FUNCTION F_ITC_SendFCR : BOOL
(**************************************************************************************
 * 	Application		:	BoxControl Framework
 *	Revision		:	$Revision: 404529 $
 *	Revision date	:	$Date: 2018-04-23 08:21:38 +0200 (Mo., 23 Apr 2018) $
 *	Last changed by	:	$Author: b7bolm $
 *	URL				:	$URL: http://almscdc.swisslog.com/repo/SWPD/Development/BoxControlFramework/20_Release/trunk/01_Software/BCF/BCF/JumpStart/20_Product/10_App/11_Com/10_Lib/10_Conv/11_ITC/F_ITC_SendFCR.TcPOU $
 *
 *	Purpose			:	Wrap message - FCR
 *
 * ------------------------------------------------------------------------------------
 *	Copyright Swisslog [IP AG], Switzerland. All rights reserved.
 * 
 * ------------------------------------------------------------------------------------
 *	
 * 	Revision History: 
 *
 * 	VERSION			DATE			INITIALS			DESCRIPTION
 *	0.1				01.01.2001		swl					Example
 *
 **************************************************************************************)
VAR_INPUT
	eChannelSrc		: E_MFCS_Channel; // Source communicaton channel	
	FunctionName	: STRING(Conveyor.POSITION_STRINGLENGTH); // The conveyor element which reports its status
	Code			: INT; // ControlCode
	Variable		: DINT; // Variable
	eReturnCode		: E_ErrorConv; // Return code
END_VAR
VAR
	FCR					: ST_ITC_FCR; 
END_VAR

// Map values
FCR.Position := FunctionName;
FCR.Code := Code;
FCR.Variable := Variable;
FCR.ReturnCode := eReturnCode;

// Forward to ITC
F_ITC_SendFCR := fbITC_Manager.M_SendData(
					meChannel	:= eChannelSrc,
					mMsgType	:= E_ITC_MsgTypeConv.FUNCTION_CONTROL_REPLY,
					mpData		:= ADR(FCR),
					mLen		:= SIZEOF(FCR));

END_FUNCTION

(* stored: Version 1.1.0.1, ProductVersion 3.1.4022.12
   POU F_ITC_SendFCR: Id {c8a45019-26c7-4f3a-bd74-3793688840a4}, SpecialFunc None *)
